// Struckig
// Copyright (C) 2022 Stefan Besler

// This program is free software: you can redistribute it and/or modify
// it under the terms of the GNU General Public License as published by
// the Free Software Foundation, either version 3 of the License, or
// (at your option) any later version.

// This program is distributed in the hope that it will be useful,
// but WITHOUT ANY WARRANTY; without even the implied warranty of
// MERCHANTABILITY or FITNESS FOR A PARTICULAR PURPOSE.  See the
// GNU General Public License for more details.
//
// You should have received a copy of the GNU General Public License
// along with THIS PROGRAM.  IF NOT, see <http://www.gnu.org/licenses/>.
/// Calculates (pre- or post-) profile to get current or final state below the limits
FUNCTION_BLOCK BrakeProfile
VAR_INPUT
  Duration : LREAL; //! Overall duration
  t, j, a, v, p : ARRAY[0..2] OF LREAL; //! Profile information for up to three-step profile  
  IsUsed : BOOL;
END_VAR
VAR
  t_to_a_min, t_to_a_max, t_min_to_v_max, t_to_a_zero, t_to_v_min, t_to_v_max : LREAL;
  t_to_v_max_with_constant, t_to_v_min_with_constant, v_at_a0, v_at_a_max, v_at_a_min : LREAL;
END_VAR

METHOD AccelerationBrake
VAR_INPUT
  v0, a0 : LREAL;
  vMax, vMin : LREAL;
  aMax, aMin : LREAL;
  jMax : LREAL;
END_VAR
j[0] := -jMax;

t_to_a_max := (a0 - aMax) / jMax;
t_to_a_zero := a0 / jMax;

v_at_a_max := VelocityAtTime(v0, a0, -jMax, t_to_a_max);
v_at_a0 := VelocityAtTime(v0, a0, -jMax, t_to_a_zero);

IF (v_at_a0 > vMax AND_THEN jMax > 0) OR_ELSE (v_at_a0 < vMax AND_THEN jMax < 0)
THEN
  VelocityBrake(v0, a0, vMax, vMin, aMax, aMin, jMax);

ELSIF (v_at_a_max < vMin AND_THEN jMax > 0) OR_ELSE (v_at_a_max > vMin AND_THEN jMax < 0)
THEN
  t_to_v_min := -(v_at_a_max - vMin)/aMax;
  t_to_v_max := -aMax/(2*jMax) - (v_at_a_max + vMax)/aMax;
  t[0] := t_to_a_max + Constants.BrakeEpsilon;
  t[1] := MAX(MIN(t_to_v_min, v_at_a_max - Constants.BrakeEpsilon), 0.0);
ELSE
  t[0] := t_to_a_max + Constants.BrakeEpsilon;
END_IF
END_METHOD

/// Finalize third-order braking by integrating along kinematic state
METHOD Finalize
VAR_IN_OUT
  ps : LREAL;
  vs : LREAL;
  as : LREAL;
END_VAR
IF t[0] <= 0 AND_THEN t[1] <= 0
THEN
  Duration := 0;
  RETURN;
END_IF

Duration := t[0];
p[0] := ps;
v[0] := vs;
a[0] := as;
Integrate(t[0], p0:=ps, v0:=vs, a0:=as, j:=j[0], p:=ps, v:=vs, a:=as);

IF t[1] > 0
THEN
  Duration := Duration + t[1];
  p[1] := ps;
  v[1] := vs;
  a[1] := as;
  Integrate(t[1], p0:=ps, v0:=vs, a0:=as, j:=j[1], p:=ps, v:=vs, a:=as);
END_IF

IF t[2] > 0
THEN
  Duration := Duration + t[2];
  p[2] := ps;
  v[2] := vs;
  a[2] := as;
  Integrate(t[2], p0:=ps, v0:=vs, a0:=as, j:=j[2], p:=ps, v:=vs, a:=as);
END_IF
END_METHOD

/// Finalize third-order braking by integrating along kinematic state
METHOD FinalizeSecondOrder
VAR_IN_OUT
  ps : LREAL;
  vs : LREAL;
  as : LREAL;
END_VAR
IF t[0] <= 0.0
THEN
  Duration := 0;
  RETURN;
END_IF

Duration := t[0];
p[0] := ps;
v[0] := vs;
Integrate(t[0], p0:=ps, v0:=vs, a0:=a[0], j:=j[0], p:=ps, v:=vs, a:=as);
END_METHOD

/// Calculate brake trajectory for third-order position interface
METHOD PositionBrakeTrajectory
VAR_INPUT
  v0, a0 : LREAL;
  vMax, vMin : LREAL;
  aMax, aMin : LREAL;
  jMax : LREAL;
  SmoothBrake : BOOL;
END_VAR
t[0] := 0.0;
t[1] := 0.0;
t[2] := 0.0;
j[0] := 0.0;
j[1] := 0.0;
j[2] := 0.0;

IF jMax = 0 OR_ELSE aMax = 0 OR_ELSE aMin = 0
THEN
  RETURN;
ELSIF a0 > aMax
THEN
  AccelerationBrake(v0, a0, vMax, vMin, aMax, aMin, jMax);
ELSIF a0 < aMin
THEN
  AccelerationBrake(v0, a0, vMin, vMax, aMin, aMax, -jMax);
ELSIF SmoothBrake AND_THEN v0 > vMax AND_THEN ABS(a0) < aMax
THEN
  SmoothVelocityBrake(v0, a0, vMax, aMax, jMax);
  IF t[0] <= 0 THEN
    VelocityBrake(v0, a0, vMax, vMin, aMax, aMin, jMax);
  END_IF
ELSIF SmoothBrake AND_THEN v0 < vMin AND_THEN ABS(a0) < aMax
THEN
  SmoothVelocityBrake(v0, a0, vMin, aMax, -jMax);
  IF t[0] <= 0 THEN
    VelocityBrake(v0, a0, vMin, vMax, aMin, aMax, -jMax);
  END_IF
ELSIF ((v0 > vMax AND_THEN VelocityAtZeroAcceleration(v0, a0, -jMax) > vMin) OR_ELSE (a0 > 0 AND_THEN VelocityAtZeroAcceleration(v0, a0, jMax) > vMax))
THEN
  VelocityBrake(v0, a0, vMax, vMin, aMax, aMin, jMax);
ELSIF ((v0 < vMin AND_THEN VelocityAtZeroAcceleration(v0, a0, jMax) < vMax) OR_ELSE (a0 < 0 AND_THEN VelocityAtZeroAcceleration(v0, a0, -jMax) < vMin))
THEN
  VelocityBrake(v0, a0, vMin, vMax, aMin, aMax, -jMax);      
END_IF
END_METHOD

/// Calculate brake trajectory for third-order position interface
METHOD SecondOrderPositionBrakeTrajectory
VAR_INPUT
  v0 : LREAL;
  vMax, vMin : LREAL;
  aMax, aMin : LREAL;
END_VAR
t[0] := 0.0;
t[1] := 0.0;
j[0] := 0.0;
j[1] := 0.0;
a[0] := 0.0;
a[1] := 0.0;

IF aMax = 0.0 OR_ELSE aMin = 0.0
THEN
  RETURN; // Ignore braking for zero-limits 
END_IF

IF v0 > vMax
THEN
  a[0] := aMin;
  t[0] := (vMax - v0)/aMin + Constants.Epsilon;   
ELSIF v0 < vMin
THEN
  a[0] := aMax;
  t[0] := (vMin - v0)/aMax + Constants.Epsilon;
END_IF
END_METHOD

/// Calculate brake trajectory for third-order position interface
METHOD SecondOrderVelocityBrakeTrajectory
VAR_INPUT
END_VAR
t[0] := 0;
t[1] := 0;
j[0] := 0;
j[1] := 0;
END_METHOD

/// Jerk-limited brake from (v0, a0) to (vTarget, a=0).
/// Produces a 2- or 3-phase profile that ends with zero acceleration,
/// so Step1 does not inherit a large residual deceleration.
/// jMax > 0 means braking from above (v0 > vTarget), jMax < 0 means from below.
/// If the profile cannot be computed (e.g. a0 opposes braking too strongly),
/// t[0] remains 0 so the caller can fall back to legacy VelocityBrake.
METHOD SmoothVelocityBrake
VAR_INPUT
  v0, a0 : LREAL;
  vTarget : LREAL;
  aMax : LREAL;
  jMax : LREAL;
END_VAR
VAR
  half_D, t1, t3, a_peak : LREAL;
  v1, dv_phase3, t2, a_clamp : LREAL;
END_VAR
IF (jMax > 0 AND_THEN v0 <= vTarget) OR_ELSE (jMax < 0 AND_THEN v0 >= vTarget) THEN
  RETURN;
END_IF

(* Solve quadratic for 2-phase brake from (v0,a0) to (vTarget,0):
   Phase 1: j = -jMax, duration t1
   Phase 3: j = +jMax, duration t3 = t1 - a0/jMax
   jMax * t1^2 - 2*a0*t1 + (vTarget - v0 + a0^2/(2*jMax)) = 0
   D/4 = a0^2/2 + jMax*(v0 - vTarget) *)
half_D := a0*a0*0.5 + jMax*(v0 - vTarget);
IF half_D < 0 THEN
  RETURN;
END_IF

IF jMax > 0 THEN
  t1 := (a0 + SQRT(half_D)) / jMax;
ELSE
  t1 := (a0 - SQRT(half_D)) / jMax;
END_IF

IF t1 < 0 THEN
  RETURN;
END_IF

t3 := t1 - a0/jMax;
a_peak := a0 - jMax*t1;

IF ABS(a_peak) <= aMax THEN
  j[0] := -jMax;
  t[0] := t1;
  j[1] := jMax;
  t[1] := t3;
  t[2] := 0;
ELSE
  (* 3-phase: clamp peak acceleration at ±aMax *)
  IF jMax > 0 THEN
    a_clamp := -aMax;
  ELSE
    a_clamp := aMax;
  END_IF

  t1 := (a0 - a_clamp) / jMax;
  t3 := -a_clamp / jMax;
  v1 := v0 + a0*t1 - 0.5*jMax*t1*t1;
  dv_phase3 := a_clamp*t3 + 0.5*jMax*t3*t3;
  t2 := (vTarget - v1 - dv_phase3) / a_clamp;

  IF t2 < 0 THEN
    RETURN;
  END_IF

  j[0] := -jMax;
  t[0] := t1;
  j[1] := 0;
  t[1] := t2;
  j[2] := jMax;
  t[2] := t3;
END_IF
END_METHOD

METHOD VelocityAtTime : LREAL
VAR_INPUT
  v0, a0 : LREAL;
  j : LREAL;
  t : LREAL;
END_VAR
VelocityAtTime := v0 + t * (a0 + j * t * 0.5);
END_METHOD

METHOD VelocityAtZeroAcceleration : LREAL
VAR_INPUT
  v0, a0 : LREAL;
  j : LREAL;
END_VAR
VelocityAtZeroAcceleration := v0 + (a0 * a0) / (2 * j);
END_METHOD

METHOD VelocityBrake
VAR_INPUT
  v0, a0 : LREAL;
  vMax, vMin : LREAL;
  aMax, aMin : LREAL;
  jMax : LREAL;
END_VAR
j[0] := -jMax;
t_to_a_min := (a0 - aMin)/jMax;
t_to_v_max := a0*a0 + 2 * jMax * (v0 - vMax);
t_to_v_min := a0*a0 / 2 + jMax * (v0 - vMin);

IF t_to_v_max < 0 OR_ELSE t_to_v_min < 0
THEN
  RETURN;
END_IF

t_to_v_max := a0/jMax + SQRT(t_to_v_max) / ABS(jMax);
t_to_v_min := a0/jMax + SQRT(t_to_v_min) / ABS(jMax);
t_min_to_v_max := MIN(t_to_v_max, t_to_v_min);

IF (t_to_a_min < t_min_to_v_max)
THEN
  v_at_a_min := VelocityAtTime(v0, a0, -jMax, t_to_a_min);
  t_to_v_max_with_constant := -(v_at_a_min - vMax)/aMin;
  t_to_v_min_with_constant := -0.5*aMin/jMax - (v_at_a_min - vMin)/aMin;
  t[0] := MAX(t_to_a_min - Constants.BrakeEpsilon, 0);
  t[1] := MAX(MIN(t_to_v_max_with_constant, t_to_v_min_with_constant), 0.0);
ELSE
  t[0] := MAX(t_min_to_v_max - Constants.BrakeEpsilon, 0);
END_IF
END_METHOD

/// Calculate brake trajectory for third-order velocity interface
METHOD VelocityBrakeTrajectory
VAR_INPUT
  v0, a0 : LREAL;
  aMax, aMin : LREAL;
  jMax : LREAL;
END_VAR
t[0] := 0.0;
t[1] := 0.0;
j[0] := 0.0;
j[1] := 0.0;

IF jMax = 0
THEN
  RETURN; // Ignore braking for zero-limits
ELSIF (a0 > aMax)
THEN
  j[0] := -jMax;
  t[0] := (a0 - aMax)/jMax + Constants.BrakeEpsilon;
ELSIF (a0 < aMin)
THEN
  j[0] := jMax;
  t[0] := -(a0 - aMin)/jMax + Constants.BrakeEpsilon;
END_IF
END_METHOD

END_FUNCTION_BLOCK

(* stored: Version 1.1.0.1
   POU BrakeProfile: Id {1eceebc8-e02e-4905-a883-8b9d67dc9558}, SpecialFunc None
   Method AccelerationBrake: Id {151af409-7ad6-4437-ae65-90af2283f00d}
   Method Finalize: Id {0fcf778f-80e5-4f55-9da3-b7c243c42728}
   Method FinalizeSecondOrder: Id {75063da7-6df2-4dc8-a3e9-7c13e02c2b78}
   Method PositionBrakeTrajectory: Id {95c53b9d-c397-464e-b5fb-c3d4cad36b7c}
   Method SecondOrderPositionBrakeTrajectory: Id {5a7eb56a-bf46-49f0-bf23-96b722fbed89}
   Method SecondOrderVelocityBrakeTrajectory: Id {50f427f5-11c2-4e9d-965a-157c6b7a0bbe}
   Method SmoothVelocityBrake: Id {d9f1a2b3-c4e5-6789-abcd-ef0123456789}
   Method VelocityAtTime: Id {f532e452-5e4d-4b4e-a9b9-55765c5c49dc}
   Method VelocityAtZeroAcceleration: Id {fadf7222-52a9-4a60-9bb7-04c04e997a4d}
   Method velocityBrake: Id {c8d0a7a0-928d-4c6d-8096-2b92af8cd1a4}
   Method VelocityBrakeTrajectory: Id {33c02e8e-5511-4646-952e-73b09c9f73ca} *)
